// TIA Portal project "prova1" (V15.1)

(* hardware
DEVICE "S7-1200 station_1"  S7-1200 Station
   slot 0: "Telaio di montaggio_0"  S7-1200 Rack  Rack  V1.0
   slot 1: "PLC_1"  CPU 1214C DC/DC/DC  6ES7 214-1AG40-0XB0  V4.2
*)

// ===== PLC "PLC_1"  CPU 1214C DC/DC/DC =====

VAR_GLOBAL   // PLC tag table "Tabella delle variabili standard"
   "L0" AT %I0.0 : Bool;
   "L1" AT %I0.1 : Bool;
   "V1" AT %I0.2 : Bool;
   "V2" AT %I0.3 : Bool;
   "MS" AT %Q0.0 : Bool;
   "MD" AT %Q0.1 : Bool;
   "Mup" AT %Q0.2 : Bool;
   "Mdown" AT %Q0.3 : Bool;
   "start" AT %I0.4 : Bool;
END_VAR

VAR_GLOBAL CONSTANT   // PLC tag table "Tabella delle variabili standard"
   "tempoAttesa" : Time := T#10s;
END_VAR

DATA_BLOCK "variabili_stato"   // DB1
{ S7_Optimized_Access := 'TRUE' }
VERSION : 0.1
   VAR RETAIN
      home : Bool := true;
      sali : Bool;
      sinistra : Bool;
      wait : Bool;
      destra : Bool;
      scendi : Bool;
   END_VAR
BEGIN
END_DATA_BLOCK

// folder: System blocks/Program resources

DATA_BLOCK "IEC_Timer_0_DB"   // DB2
{ S7_Optimized_Access := 'TRUE' }
AUTHOR : Simatic
FAMILY : IEC
NAME : IEC_TMR
VERSION : 1.0
// stored: InstanceOfName IEC_TIMER
"IEC_TIMER"
BEGIN
END_DATA_BLOCK

// folder: (top level)

ORGANIZATION_BLOCK "Main"   // OB1, LAD, ProgramCycle
TITLE = "Main Program Sweep (Cycle)"
{ S7_Optimized_Access := 'TRUE' }
VERSION : 0.1
   VAR_INPUT
      Initial_Call : Bool;   // Initial call of this OB
      Remanence : Bool;   // =True, if remanent data are available
   END_VAR
   VAR_TEMP
      temp : Bool;
   END_VAR
   VAR_TEMP   // added for the SCL form of the ladder/FBD networks
      _w1 : Bool;
   END_VAR
BEGIN

REGION Network 1
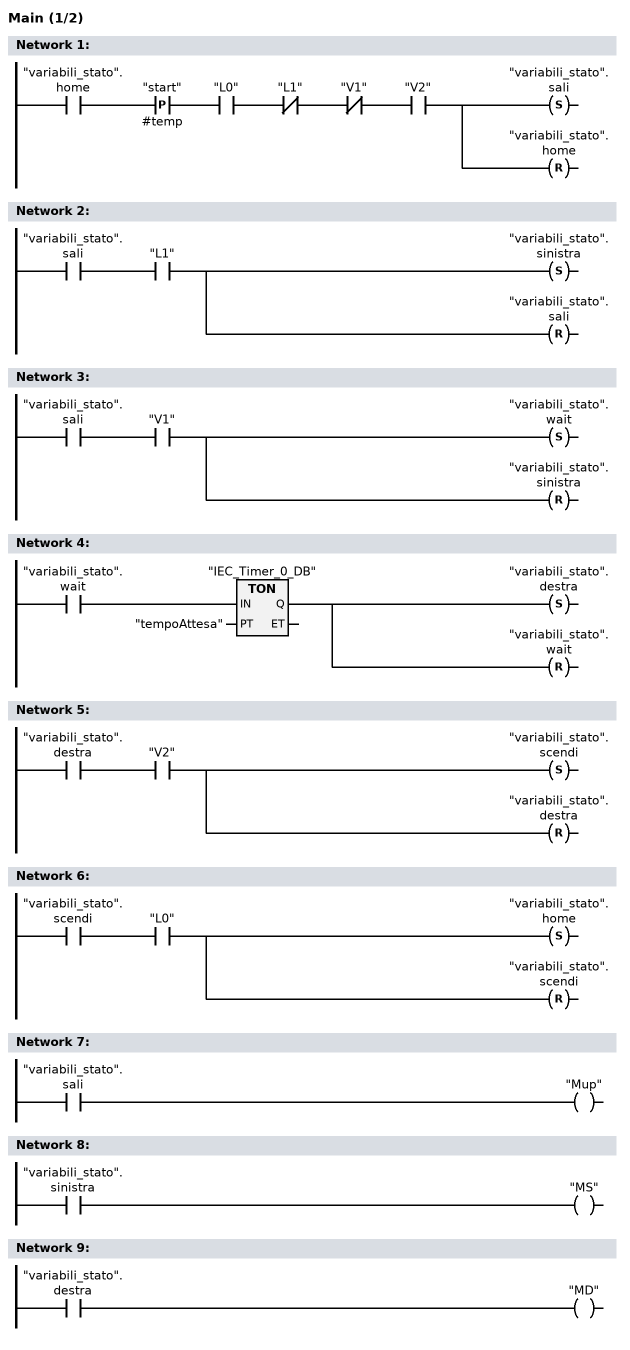
   RUNG wire#powerrail
      Contact( "variabili_stato".home )
      P_Contact(operand := "start", bit := #temp)
      Contact( "L0" )
      I_Contact( "L1" )
      I_Contact( "V1" )
      Contact( "V2" )
      wire#w1
      S_Coil( "variabili_stato".sali )
   END_RUNG
   RUNG wire#w1
      R_Coil( "variabili_stato".home )
   END_RUNG
   // the same network as SCL:
   #_w1 := "variabili_stato".home AND "start" AND NOT #temp;   // rising edge of "start"
   #temp := "start";
   IF #_w1 AND "L0" AND NOT "L1" AND NOT "V1" AND "V2" THEN
       "variabili_stato".sali := TRUE;
       "variabili_stato".home := FALSE;
   END_IF;
END_REGION

REGION Network 2
   RUNG wire#powerrail
      Contact( "variabili_stato".sali )
      Contact( "L1" )
      wire#w1
      S_Coil( "variabili_stato".sinistra )
   END_RUNG
   RUNG wire#w1
      R_Coil( "variabili_stato".sali )
   END_RUNG
   // the same network as SCL:
   IF "variabili_stato".sali AND "L1" THEN
       "variabili_stato".sinistra := TRUE;
       "variabili_stato".sali := FALSE;
   END_IF;
END_REGION

REGION Network 3
   RUNG wire#powerrail
      Contact( "variabili_stato".sali )
      Contact( "V1" )
      wire#w1
      S_Coil( "variabili_stato".wait )
   END_RUNG
   RUNG wire#w1
      R_Coil( "variabili_stato".sinistra )
   END_RUNG
   // the same network as SCL:
   IF "variabili_stato".sali AND "V1" THEN
       "variabili_stato".wait := TRUE;
       "variabili_stato".sinistra := FALSE;
   END_IF;
END_REGION

REGION Network 4
   "IEC_Timer_0_DB".TON(IN := "variabili_stato".wait, PT := "tempoAttesa");
   IF "IEC_Timer_0_DB".Q THEN
       "variabili_stato".destra := TRUE;
       "variabili_stato".wait := FALSE;
   END_IF;
END_REGION

REGION Network 5
   RUNG wire#powerrail
      Contact( "variabili_stato".destra )
      Contact( "V2" )
      wire#w1
      S_Coil( "variabili_stato".scendi )
   END_RUNG
   RUNG wire#w1
      R_Coil( "variabili_stato".destra )
   END_RUNG
   // the same network as SCL:
   IF "variabili_stato".destra AND "V2" THEN
       "variabili_stato".scendi := TRUE;
       "variabili_stato".destra := FALSE;
   END_IF;
END_REGION

REGION Network 6
   RUNG wire#powerrail
      Contact( "variabili_stato".scendi )
      Contact( "L0" )
      wire#w1
      S_Coil( "variabili_stato".home )
   END_RUNG
   RUNG wire#w1
      R_Coil( "variabili_stato".scendi )
   END_RUNG
   // the same network as SCL:
   IF "variabili_stato".scendi AND "L0" THEN
       "variabili_stato".home := TRUE;
       "variabili_stato".scendi := FALSE;
   END_IF;
END_REGION

REGION Network 7
   RUNG wire#powerrail
      Contact( "variabili_stato".sali )
      Coil( "Mup" )
   END_RUNG
   // the same network as SCL:
   "Mup" := "variabili_stato".sali;
END_REGION

REGION Network 8
   RUNG wire#powerrail
      Contact( "variabili_stato".sinistra )
      Coil( "MS" )
   END_RUNG
   // the same network as SCL:
   "MS" := "variabili_stato".sinistra;
END_REGION

REGION Network 9
   RUNG wire#powerrail
      Contact( "variabili_stato".destra )
      Coil( "MD" )
   END_RUNG
   // the same network as SCL:
   "MD" := "variabili_stato".destra;
END_REGION

REGION Network 10
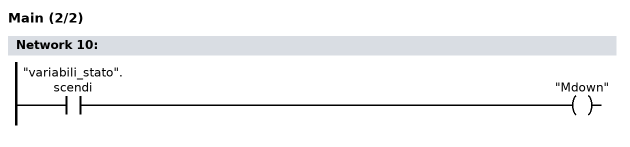
   RUNG wire#powerrail
      Contact( "variabili_stato".scendi )
      Coil( "Mdown" )
   END_RUNG
   // the same network as SCL:
   "Mdown" := "variabili_stato".scendi;
END_REGION
END_ORGANIZATION_BLOCK